// TIA Portal V20 export
TYPE "typeEm2Monitoring"
// stored: Access Published, Namespace Unit1
   STRUCT
      jobinterface { ExternalWritable := 'False'} : "Unit1.typeEm2MonitoringJobInterface";
      cmStatus { ExternalWritable := 'False'} : "Unit1.typeEm2MonitoringCmStatus";
      UserDefine { ExternalWritable := 'False'} : "Unit1.typeEm2MonitoringUserDefine";
   END_STRUCT;
END_TYPE
